// TIA Portal project "Training" (V13)

(* hardware
DEVICE "S71500/ET200MP station_1"  S7-1500 station
   slot 0: "Rail_0"  6ES7 590-1***0-0AA0
   slot 1: "PLC_1"  CPU 1516F-3 PN/DP  6ES7 516-3FN00-0AB0  V1.7
   slot 2: "DI 16x24VDC HF_1"  DI 16x24VDC HF  6ES7 521-1BH00-0AB0  V2.0
   slot 3: "AI 8xU/I/RTD/TC ST_1"  AI 8xU/I/RTD/TC ST  6ES7 531-7KF00-0AB0  V2.0
   slot 4: "CP 1543-1_1"  CP 1543-1  6GK7 543-1AX00-0XE0  V1.1
*)

// ===== PLC "PLC_1"  CPU 1516F-3 PN/DP =====

VAR_GLOBAL   // PLC tag table "Default tag table"
   "System_Byte" AT %MB1 : Byte;
   "FirstScan" AT %M1.0 : Bool;
   "DiagStatusUpdate" AT %M1.1 : Bool;
   "AlwaysTRUE" AT %M1.2 : Bool;
   "AlwaysFALSE" AT %M1.3 : Bool;
   "Clock_Byte" AT %MB0 : Byte;
   "Clock_10Hz" AT %M0.0 : Bool;
   "Clock_5Hz" AT %M0.1 : Bool;
   "Clock_2.5Hz" AT %M0.2 : Bool;
   "Clock_2Hz" AT %M0.3 : Bool;
   "Clock_1.25Hz" AT %M0.4 : Bool;
   "Clock_1Hz" AT %M0.5 : Bool;
   "Clock_0.625Hz" AT %M0.6 : Bool;
   "Clock_0.5Hz" AT %M0.7 : Bool;
   "Latch Output" AT %Q50.0 : Bool;
   "Indicated Deg C_1" AT %MW2 : Int;
   "Indicated Deg c_2" AT %MW4 : Int;
   "Run Status" AT %M6.0 : Bool;
   "Counter Reset Bit" AT %M6.1 : Bool;
   "Motor 1 Running" AT %M6.2 : Bool;
   "Motor 2 Running" AT %M6.3 : Bool;
END_VAR

VAR_GLOBAL   // PLC tag table "Local IO Tags"
   "S71500 Green PB" AT %I0.0 : Bool;
   "S71500 Blue PB" AT %I0.1 : Bool;
   "S71500 Pot Upper" AT %IW6 : Int;
   "S71500 Pot Lower" AT %IW14 : Int;
END_VAR

TYPE "Motor Control"
   STRUCT
      "Motor Start/Stop" : Bool;
      "Motor Run" : Bool;
      "Counter Reset" : Bool;
      "Count Value" : Int;
   END_STRUCT;
END_TYPE

DATA_BLOCK "My Global Data"   // DB1
{ S7_Optimized_Access := 'FALSE' }
VERSION : 0.1
   VAR
      "Celsius Temperature 1" : Int;
      "Celsius Temperature 2" : Int;
      "My INT Value" : Int;
      "My INT Setpoint Value" : Int;
   END_VAR
BEGIN
END_DATA_BLOCK

DATA_BLOCK "FB Motor Starter_DB"   // DB2
{ S7_Optimized_Access := 'FALSE' }
VERSION : 0.1
// stored: InstanceOfName FB Motor Starter
"FB Motor Starter"
BEGIN
END_DATA_BLOCK

DATA_BLOCK "FB Motor Controls_DB"   // DB3
{ S7_Optimized_Access := 'FALSE' }
VERSION : 0.1
// stored: InstanceOfName FB Motor Controls
"FB Motor Controls"
BEGIN
END_DATA_BLOCK

DATA_BLOCK "DB Motor Controls"   // DB4
{ S7_Optimized_Access := 'FALSE' }
VERSION : 0.1
   VAR
      Motor : Array[1..2] of "Motor Control";
   END_VAR
BEGIN
END_DATA_BLOCK

DATA_BLOCK "FB Motor Controls_DB_1"   // DB5
{ S7_Optimized_Access := 'FALSE' }
VERSION : 0.1
// stored: InstanceOfName FB Motor Controls
"FB Motor Controls"
BEGIN
END_DATA_BLOCK

FUNCTION_BLOCK "FB Motor Starter"   // FB1, LAD
{ S7_Optimized_Access := 'FALSE' }
VERSION : 0.1
   VAR_TEMP   // added for the SCL form of the ladder/FBD networks
      _w1 : Bool;
      _w2 : Bool;
   END_VAR
BEGIN

REGION Network 1
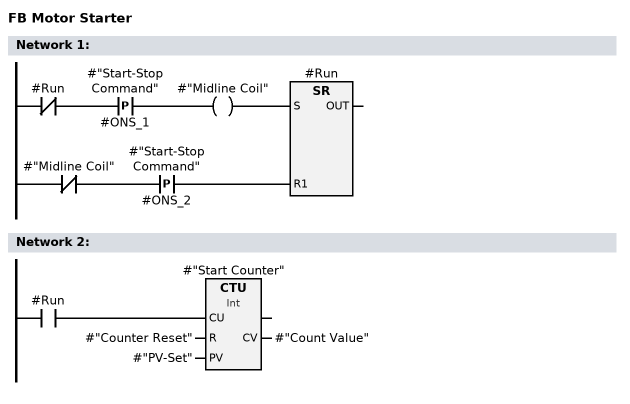
   RUNG wire#powerrail
      I_Contact( #Run )
      P_Contact(operand := #"Start-Stop Command", bit := #ONS_1)
      Coil( #"Midline Coil" )
      S_SR(operand := #Run, r1 := wire#w1)
   END_RUNG
   RUNG wire#powerrail
      I_Contact( #"Midline Coil" )
      P_Contact(operand := #"Start-Stop Command", bit := #ONS_2)
   END_RUNG wire#w1
   // the same network as SCL:
   #_w1 := NOT #Run AND #"Start-Stop Command" AND NOT #ONS_1;   // rising edge of #"Start-Stop Command"
   #ONS_1 := #"Start-Stop Command";
   #"Midline Coil" := #_w1;
   #_w2 := NOT #"Midline Coil" AND #"Start-Stop Command" AND NOT #ONS_2;   // rising edge of #"Start-Stop Command"
   #ONS_2 := #"Start-Stop Command";
   IF #_w1 THEN
       #Run := TRUE;   // SR flip-flop
   END_IF;
   IF #_w2 THEN #Run := FALSE; END_IF;
END_REGION

REGION Network 2
   #"Start Counter".CTU(CU := #Run, R := #"Counter Reset", PV := #"PV-Set", CV => #"Count Value");
END_REGION
END_FUNCTION_BLOCK

FUNCTION_BLOCK "FB Motor Controls"   // FB2, LAD
{ S7_Optimized_Access := 'FALSE' }
VERSION : 0.1
BEGIN

REGION Network 1
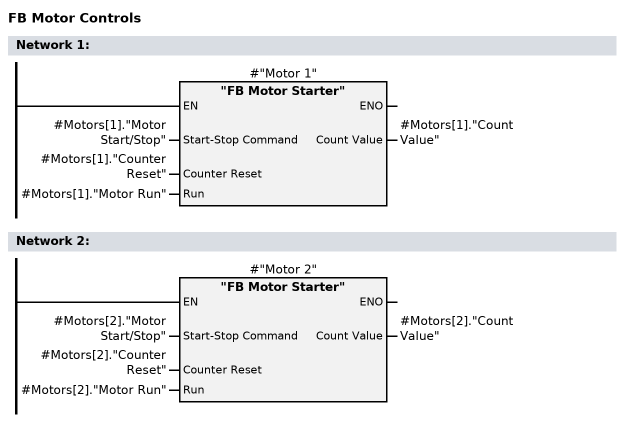
   RUNG wire#powerrail
      #"Motor 1"("Start-Stop Command" := #Motors[1]."Motor Start/Stop", "Counter Reset" := #Motors[1]."Counter Reset", Run := #Motors[1]."Motor Run", "Count Value" => #Motors[1]."Count Value")
   END_RUNG
   // the same network as SCL:
   #"Motor 1"("Start-Stop Command" := #Motors[1]."Motor Start/Stop",   // "FB Motor Starter"
              "Counter Reset" := #Motors[1]."Counter Reset",
              Run := #Motors[1]."Motor Run",
              "Count Value" => #Motors[1]."Count Value");
END_REGION

REGION Network 2
   RUNG wire#powerrail
      #"Motor 2"("Start-Stop Command" := #Motors[2]."Motor Start/Stop", "Counter Reset" := #Motors[2]."Counter Reset", Run := #Motors[2]."Motor Run", "Count Value" => #Motors[2]."Count Value")
   END_RUNG
   // the same network as SCL:
   #"Motor 2"("Start-Stop Command" := #Motors[2]."Motor Start/Stop",   // "FB Motor Starter"
              "Counter Reset" := #Motors[2]."Counter Reset",
              Run := #Motors[2]."Motor Run",
              "Count Value" => #Motors[2]."Count Value");
END_REGION
END_FUNCTION_BLOCK

FUNCTION "F to C Conversion" : Void   // FC1, LAD
{ S7_Optimized_Access := 'FALSE' }
VERSION : 0.1
BEGIN

REGION Network 1
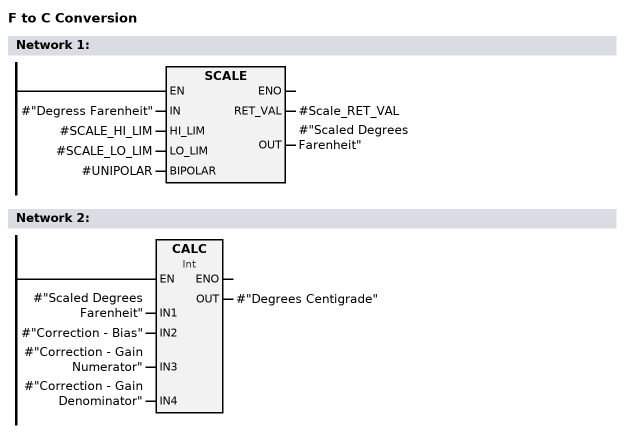
   #Scale_RET_VAL := SCALE(IN := #"Degress Farenheit",
                           HI_LIM := #SCALE_HI_LIM,
                           LO_LIM := #SCALE_LO_LIM,
                           BIPOLAR := #UNIPOLAR,
                           OUT => #"Scaled Degrees Farenheit");
END_REGION

REGION Network 2
   CALC(in1 := #"Scaled Degrees Farenheit",
        in2 := #"Correction - Bias",
        in3 := #"Correction - Gain Numerator",
        in4 := #"Correction - Gain Denominator",
        out => #"Degrees Centigrade");
END_REGION
END_FUNCTION

ORGANIZATION_BLOCK "Main"   // OB1, LAD, ProgramCycle
TITLE = "Main Program Sweep (Cycle)"
{ S7_Optimized_Access := 'FALSE' }
VERSION : 0.1
BEGIN

REGION Network 1
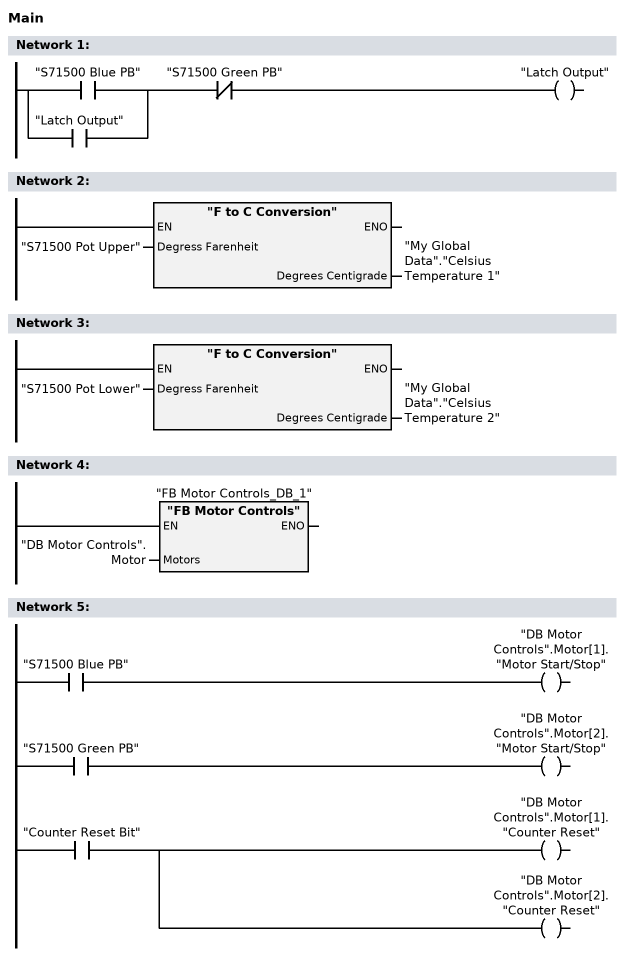
   RUNG wire#powerrail
      Contact( "S71500 Blue PB" )
      wire#w1
      I_Contact( "S71500 Green PB" )
      Coil( "Latch Output" )
   END_RUNG
   RUNG wire#powerrail
      Contact( "Latch Output" )
   END_RUNG wire#w1
   // the same network as SCL:
   "Latch Output" := ("S71500 Blue PB" OR "Latch Output") AND NOT "S71500 Green PB";
END_REGION

REGION Network 2
   RUNG wire#powerrail
      "F to C Conversion"("Degress Farenheit" := "S71500 Pot Upper", "Degrees Centigrade" => "My Global Data"."Celsius Temperature 1")
   END_RUNG
   // the same network as SCL:
   "F to C Conversion"("Degress Farenheit" := "S71500 Pot Upper",
                       "Degrees Centigrade" => "My Global Data"."Celsius Temperature 1");
END_REGION

REGION Network 3
   RUNG wire#powerrail
      "F to C Conversion"("Degress Farenheit" := "S71500 Pot Lower", "Degrees Centigrade" => "My Global Data"."Celsius Temperature 2")
   END_RUNG
   // the same network as SCL:
   "F to C Conversion"("Degress Farenheit" := "S71500 Pot Lower",
                       "Degrees Centigrade" => "My Global Data"."Celsius Temperature 2");
END_REGION

REGION Network 4
   RUNG wire#powerrail
      "FB Motor Controls_DB_1"(Motors := "DB Motor Controls".Motor)
   END_RUNG
   // the same network as SCL:
   "FB Motor Controls_DB_1"(Motors := "DB Motor Controls".Motor);   // "FB Motor Controls"
END_REGION

REGION Network 5
   RUNG wire#powerrail
      Contact( "S71500 Blue PB" )
      Coil( "DB Motor Controls".Motor[1]."Motor Start/Stop" )
   END_RUNG
   RUNG wire#powerrail
      Contact( "S71500 Green PB" )
      Coil( "DB Motor Controls".Motor[2]."Motor Start/Stop" )
   END_RUNG
   RUNG wire#powerrail
      Contact( "Counter Reset Bit" )
      wire#w1
      Coil( "DB Motor Controls".Motor[1]."Counter Reset" )
   END_RUNG
   RUNG wire#w1
      Coil( "DB Motor Controls".Motor[2]."Counter Reset" )
   END_RUNG
   // the same network as SCL:
   "DB Motor Controls".Motor[1]."Motor Start/Stop" := "S71500 Blue PB";
   "DB Motor Controls".Motor[2]."Motor Start/Stop" := "S71500 Green PB";
   "DB Motor Controls".Motor[1]."Counter Reset" := "Counter Reset Bit";
   "DB Motor Controls".Motor[2]."Counter Reset" := "Counter Reset Bit";
END_REGION
END_ORGANIZATION_BLOCK